// TIA Portal V19 program export: 1 tag tables, 0 data types, 0 data blocks, 3 code blocks (in call order from the OBs), 1 instance data blocks

VAR_GLOBAL   // PLC tag table "Default tag table"
   Tag_1 AT %M0.0 : Bool;
   NOWE_TAGSY AT %M0.1 : Bool;
END_VAR

ORGANIZATION_BLOCK "MainOB"   // OB1, LAD, ProgramCycle
TITLE = "Main Program Sweep (Cycle)"
{ S7_Optimized_Access := 'TRUE' }
// stored: SetENOAutomatically false
   VAR_INPUT
      Initial_Call : Bool;   // Initial call of this OB
      Remanence : Bool;   // =True, if remanent data are available
   END_VAR
   VAR_TEMP   // added for the SCL form of the ladder/FBD networks
      _w1 : Bool;
   END_VAR
BEGIN

REGION Network 1
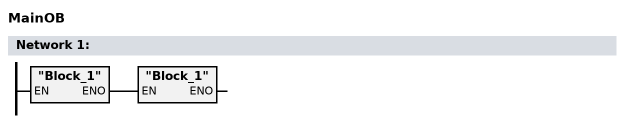
   RUNG wire#powerrail
      "Block_1"()
      "Block_1"()
   END_RUNG
   // the same network as SCL:
   "Block_1"(ENO => #_w1);
   IF #_w1 THEN "Block_1"(); END_IF;
END_REGION
END_ORGANIZATION_BLOCK

FUNCTION "Block_1" : Void   // FC1, LAD
{ S7_Optimized_Access := 'TRUE' }
// stored: SetENOAutomatically false
BEGIN
END_FUNCTION

FUNCTION "Block_2" : Void   // FC2, LAD
{ S7_Optimized_Access := 'TRUE' }
// stored: SetENOAutomatically false
BEGIN
END_FUNCTION

DATA_BLOCK "SIMATIC Ident_1"   // DB1
AUTHOR : SIMATIC
FAMILY : Ident
VERSION : 1.2
// stored: InstanceOfName TO_IDENT, OfSystemLibElement TO_IDENT, OfSystemLibVersion 1.2
TO_IDENT   // technology object, version 1.2
   // VAR
   //    HW_ID { ExternalWritable := 'False'; S7_SetPoint := 'True'} : Word;
   //    CM_CHANNEL { ExternalWritable := 'False'; S7_SetPoint := 'True'} : Int;
   //    LADDR { ExternalWritable := 'False'; S7_SetPoint := 'True'} : Word;
   //    CONFIGURATION { S7_SetPoint := 'True'} : IID_IN_PARAMETERS;
   //    DIAGNOSTIC { ExternalWritable := 'False'; S7_SetPoint := 'True'} : IID_IN_DIAGNOSTIC;
   //    STATIC { ExternalWritable := 'False'; S7_SetPoint := 'True'} : IID_IN_SYNC_TO;
   // END_VAR
BEGIN
END_DATA_BLOCK
